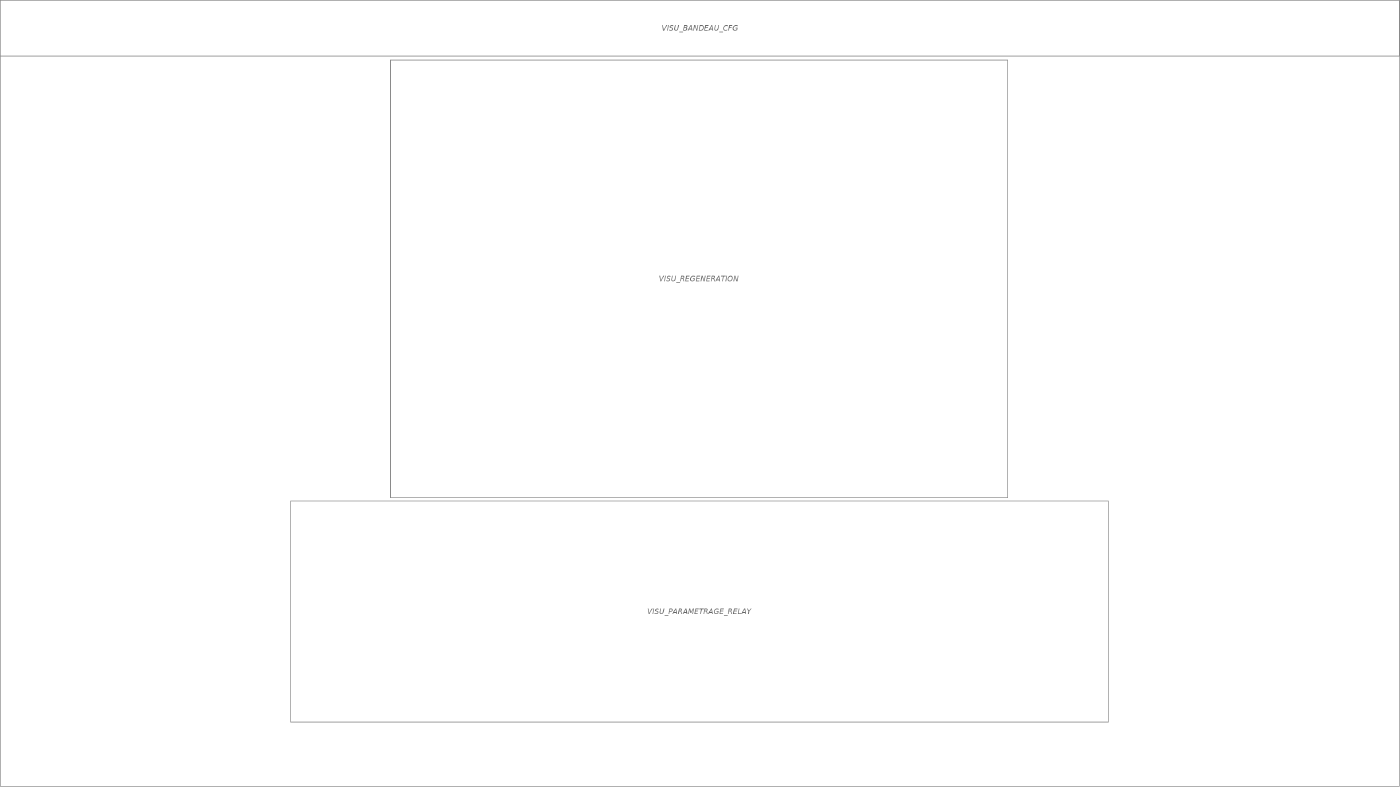
VISUALIZATION VISU_CONFIG_REGEN  // 1920x1080, background image fond_blanc_1280_1024
    Frame (0,0 1920x77)
        shows VISU_BANDEAU_CFG()
    Frame (535,82 847x601)
        shows VISU_REGENERATION(COM := PRG_POMPAGE.COM_CRYOS)
    Frame (398,687 1122x304)
        shows VISU_PARAMETRAGE_RELAY(COM := PRG_POMPAGE.COM_CRYOS)
END_VISUALIZATION

(* stored: Version 1.1.0.1, ProductVersion 3.1.4026.18
   Visu VISU_CONFIG_REGEN: Id {57168ad9-7c75-43fe-8a6a-ca9c40f5573b} *)
